PROGRAM MAIN
VAR
END_VAR

END_PROGRAM

(* stored: Version 1.1.0.1
   POU MAIN: Id {1afdb442-89ec-4be5-b36d-4b87f4b5924f} *)
